{attribute 'linkalways'} 
{attribute 'no_explicit_call' := 'This FB is a CLASS and must be accessed using methods or properties'}
{attribute 'enable_dynamic_creation'}
FUNCTION_BLOCK _ETcVnDistanceTransformationLabel EXTENDS EnumDatatypeBase
VAR
	localData : ETcVnDistanceTransformationLabel;
	activeData : REFERENCE TO ETcVnDistanceTransformationLabel;
	enumBaseDatatype : _DINT(localData);
END_VAR

METHOD PRIVATE AddLocalEnumeration
VAR_INPUT
	Enumeration : T_MAXSTRING;
	Value : ETcVnDistanceTransformationLabel;
END_VAR
AddEnumeration(Enumeration, Value);
END_METHOD

PROPERTY PUBLIC Address : PVOID
GET
Address := ADR(activeData);
END_GET
END_PROPERTY

METHOD PUBLIC ClearReference
VAR_INPUT
END_VAR
activeData REF= localData;
SetBaseDatatypeReference();
END_METHOD

METHOD PUBLIC Clone : I_Datatype
VAR
    pClone : POINTER TO _ETcVnDistanceTransformationLabel;
END_VAR
pClone := __NEW(_ETcVnDistanceTransformationLabel(InitialValue := Value));
Clone := pClone^;
END_METHOD

METHOD FB_init : BOOL
VAR_INPUT
	bInitRetains : BOOL; // if TRUE, the retain variables are initialized (warm start / cold start)
	bInCopyCode : BOOL;  // if TRUE, the instance afterwards gets moved into the copy code (online change)
	InitialValue : ETcVnDistanceTransformationLabel;
END_VAR
localData := InitialValue;
AddBaseDatatype(enumBaseDatatype);
ClearReference();

AddLocalEnumeration('TCVN_DTL_CCOMP', ETcVnDistanceTransformationLabel.TCVN_DTL_CCOMP);
AddLocalEnumeration('TCVN_DTL_PIXEL', ETcVnDistanceTransformationLabel.TCVN_DTL_PIXEL);
END_METHOD

PROPERTY PUBLIC Identifier : T_MAXSTRING
GET
Identifier := 'ETcVnDistanceTransformationLabel';
END_GET
END_PROPERTY

METHOD IsEnumeratorValueEqual : BOOL
VAR_INPUT
	Enumerator : I_KeyValueForwardEnumerator;
END_VAR
VAR
	storedValue : ETcVnDistanceTransformationLabel;
END_VAR
IF NOT Enumerator.TryGet(storedValue) THEN
	RETURN;
END_IF

IsEnumeratorValueEqual := storedValue = activeData;
END_METHOD

METHOD PUBLIC MakeReferenceTo
VAR_INPUT
	ReferenceTarget : REFERENCE TO ETcVnDistanceTransformationLabel;
END_VAR
activeData REF= ReferenceTarget;
SetBaseDatatypeReference();
END_METHOD

METHOD PROTECTED SetBaseDatatypeReference
VAR_INPUT
END_VAR
enumBaseDatatype.MakeReferenceTo(activeData);
END_METHOD

PROPERTY PUBLIC Size : UDINT
GET
Size := SIZEOF(activeData);
END_GET
END_PROPERTY

METHOD TryMakeReferenceTo : BOOL
VAR_INPUT
	Target : I_Datatype;
END_VAR
VAR
	targetAsEnum : I_EnumDatatype;
	pTargetData : POINTER TO ETcVnDistanceTransformationLabel;
END_VAR
IF NOT Target.TryResolveAsEnumDatatype(targetAsEnum) THEN
	RETURN;
END_IF

IF targetAsEnum.Identifier <> Identifier THEN
	RETURN;
END_IF

pTargetData := Target.Address;
activeData REF= pTargetData^;
SetBaseDatatypeReference();
TryMakeReferenceTo := TRUE;
END_METHOD

PROPERTY PUBLIC Value : ETcVnDistanceTransformationLabel
GET
Value := activeData;
END_GET
SET
activeData := Value;
END_SET
END_PROPERTY

END_FUNCTION_BLOCK

(* stored: Version 1.1.0.1
   POU _ETcVnDistanceTransformationLabel: Id {a2a021de-92a2-4e99-bd06-28462f1dd348}, SpecialFunc None
   Folder Constructor: Id {668a20f3-eab7-4715-8003-e0adef981c21}
   Folder Private: Id {c51b3296-e08e-41e5-834c-060bb15cecad}
   Folder Protected: Id {13693cb2-d9df-44ed-b6a6-c3cce610989b}
   Method AddLocalEnumeration: Id {5f8a4689-2926-440e-a42a-c3bc0ae01391}
   Property Address: Id {e8b5f5b9-f3c1-44f3-a274-5bee9d142590}
   Get Get: Id {06b8728d-07a4-47ad-8745-5039027b6352}
   Method ClearReference: Id {498b4bbb-f572-440b-bbd1-5bb1fa769554}
   Method Clone: Id {3eac0ef3-9b8b-4647-bb12-296052e2ed04}
   Method FB_init: Id {60cb4f9c-9572-4926-b8fa-d951864b1a78}
   Property Identifier: Id {bd6452a6-e8cc-4681-941c-897aff2192c8}
   Get Get: Id {f538a0c5-2dac-45d2-83a0-bc8ff501336d}
   Method IsEnumeratorValueEqual: Id {e42894b3-eb9f-44d8-9ea7-93b45bf6ecbd}
   Method MakeReferenceTo: Id {82bd5d3d-b048-4777-a944-a736ced72a49}
   Method SetBaseDatatypeReference: Id {adc8e704-5b69-4d89-8935-f9f042cb02a6}
   Property Size: Id {4417e59b-2115-48c9-96ad-6478a11c7cf8}
   Get Get: Id {b9f6e970-bdfd-42af-b5a0-50c3494ea2e6}
   Method TryMakeReferenceTo: Id {09be8118-aeda-4282-a791-715f9ca53a20}
   Property Value: Id {8d84550b-fe29-43a5-a4c3-8c71544124c7}
   Get Get: Id {68c40354-4cfa-4afd-858e-90c5ee7e90d0}
   Set Set: Id {e75041c2-c1da-4bc8-b229-a552473880b7} *)
